PROGRAM INDEXING_2
VAR
	bStartInput : BOOL;
	bServoOn : BOOL;
	bProgram0_On : BOOL;
	bProgram1_On : BOOL :=TRUE;
	bProgram2_On : BOOL :=FALSE;
	bProgram3_On : BOOL:=FALSE;
	bProgram4_On : BOOL:=FALSE;	
	bHomePositionReturn : BOOL;
	bResetInput : BOOL;
	bEmergencyInput : BOOL := TRUE;
	
	IN_POSITION_INPUT: BOOL;
	IN_POSITIONING_COMPLETION: BOOL;
	IN_START_INPUT_WAIT: BOOL;
	IN_ALARM1: BOOL;
	IN_ALARM2: BOOL;
	IN_READY_STATE: BOOL;
	T1: TON;
	TMR1: TON;
	TMR2: TON;
	TMR3: TON;
	TMR4: TON;
	TMR5: TON;
	TMR6: TON;
	TMR7: TON;
	IN_SERVO_STATUS: BOOL;
	CNT1: CTU;
	ENABLE_TIMER: INT;
	ResetCount: BOOL;
	CNT_INDEX: CTU;
	
	RESET_CNT_INDEX: BOOL;
	TMR8: TON;
	M1:BOOL;
	M2:BOOL;
	M3:BOOL;
	M4:BOOL;
	TMR_OFF: TON;
	TMR_RELEASE: TON;
	IDX: INT;
END_VAR

VAR CONSTANT
	ISP: R_TRIG;
END_VAR

INDEXING_2_VAR.DataByteOutput2[0].0 := bProgram0_On;
INDEXING_2_VAR.DataByteOutput2[0].1 := bProgram1_On;
INDEXING_2_VAR.DataByteOutput2[0].2 := bProgram2_On;
INDEXING_2_VAR.DataByteOutput2[0].3 := bProgram3_On;
INDEXING_2_VAR.DataByteOutput2[0].4 := bProgram4_On;
INDEXING_2_VAR.DataByteOutput2[0].6 := bResetInput;
INDEXING_2_VAR.DataByteOutput2[0].7 := bHomePositionReturn;
INDEXING_2_VAR.DataByteOutput2[1].0 := bStartInput;
INDEXING_2_VAR.DataByteOutput2[1].1 := bServoOn;
INDEXING_2_VAR.DataByteOutput2[1].4 := bEmergencyInput;

IN_POSITION_INPUT := INDEXING_2_VAR.DataByteInput2 [1].0;
IN_POSITIONING_COMPLETION := INDEXING_2_VAR.DataByteInput2 [1].1;
IN_START_INPUT_WAIT := INDEXING_2_VAR.DataByteInput2 [1].2;
IN_ALARM1 := INDEXING_2_VAR.DataByteInput2 [1].3;
IN_ALARM2 := INDEXING_2_VAR.DataByteInput2 [1].4;
IN_READY_STATE :=INDEXING_2_VAR.DataByteInput2 [1].7;
IN_SERVO_STATUS :=INDEXING_2_VAR.DataByteInput2 [1].6; 

M1:=INDEXING_2_VAR.DataByteInput2 [0].0;
M2:=INDEXING_2_VAR.DataByteInput2 [0].1;
M3:=INDEXING_2_VAR.DataByteInput2 [0].2;
M4:=INDEXING_2_VAR.DataByteInput2 [0].3;
bProgram1_On:=FALSE;
bProgram2_On:=FALSE;
bProgram3_On:=FALSE;
bProgram4_On:=FALSE;

//CEK SERVO STATUS
IF NOT IN_SERVO_STATUS THEN
	bResetInput := TRUE;
	TMR4(IN:=bResetInput,PT:=T#0.5S);
	IF TMR4.Q THEN
		bResetInput := FALSE;
	END_IF
	bServoOn:=TRUE;
	//POWER_CONTROL.O_PWR_CTRL_INDEXING_2:=TRUE;
	TMR8(IN:=POWER_CONTROL.O_PWR_CTRL_INDEXING_2,PT:=T#0.5S);	
	IF TMR8.Q THEN
		POWER_CONTROL.O_PWR_CTRL_INDEXING_2:=FALSE;
		TMR8(IN:=FALSE);
	END_IF
END_IF

//ALARM RESET
IF NOT IN_ALARM1 OR NOT IN_ALARM2 THEN
	bResetInput := TRUE;
	TMR4(IN:=bResetInput,PT:=T#0.5S);
		INPUT_VAR.ALARM1:=NOT IN_ALARM1 OR NOT IN_ALARM2;
	IF TMR4.Q THEN
		bResetInput := FALSE;
	END_IF
ELSE
	TMR4(IN:=FALSE);
END_IF

//HOMING
IF NOT INDEXING_2_VAR.I_INDEXING_2_HOME THEN
 	INDEXING_2_VAR.O_INDEXING_HOME:=TRUE;
END_IF
 
IF INDEXING_2_VAR.O_INDEXING_HOME THEN
	bHomePositionReturn:=TRUE;
	ResetCount:=TRUE;
	INDEXING_2_VAR.I_INDEXING_2_ROTATION_DONE:=FALSE;
	RESET_CNT_INDEX:=TRUE;
ELSE
	RESET_CNT_INDEX:=FALSE;
	bHomePositionReturn:=FALSE;
END_IF

ISP(CLK:=IN_POSITIONING_COMPLETION);	
IF 	ISP.Q THEN
	INDEXING_2_VAR.I_INDEXING_2_ROTATION_DONE:=TRUE;
END_IF

IF INDEXING_2_VAR.I_INDEXING_2_ROTATION_DONE OR INDEXING_2_VAR.O_ROTATION_DONE THEN
	INDEXING_2_VAR.I_INDEXING_2_HOME:=TRUE;
	INDEXING_2_VAR.O_INDEXING_HOME:=FALSE;
END_IF
//POWER RESET
IF bHomePositionReturn OR NOT INDEXING_2_VAR.I_INDEXING_2_ROTATION_DONE THEN
	TMR_OFF(IN:=TRUE,PT:=T#60S);
	IF TMR_OFF.Q THEN
		POWER_CONTROL.O_PWR_CTRL_INDEXING_2:=TRUE;
		TMR_RELEASE(IN:=TRUE,PT:=T#0.5S);
		BPROGRAM0_ON:=FALSE;
	END_IF
ELSE
	TMR_OFF(IN:=FALSE);
	TMR_RELEASE(IN:=FALSE);
END_IF

IF TMR_RELEASE.Q THEN
	POWER_CONTROL.O_PWR_CTRL_INDEXING_1:=FALSE;
	TMR_OFF(IN:=FALSE);
END_IF



//START ROTATION 
	IF 	INDEXING_2_VAR.O_ROTATION_START AND IN_START_INPUT_WAIT AND NOT INDEXING_2_VAR.O_INDEXING_HOME THEN
		IDX:=1;
		INDEXING_2_VAR.I_INDEXING_2_ROTATION_DONE:=FALSE;
	END_IF
CASE IDX OF
1:
	bprogram0_on:=TRUE;
	IF BPROGRAM0_ON THEN
		IDX:=2;
		INDEXING_2_VAR.O_ROTATION_START:=FALSE;
	END_IF

2:
//select Program No.
	IF bprogram0_on THEN
		INDEXING_2_VAR.O_ROTATION_START:=FALSE;
		INDEXING_2_VAR.I_INDEXING_2_ROTATION_DONE:=FALSE;
		TMR1(IN:=bprogram0_on,PT:=T#15MS);
		bStartInput:=tmr1.Q ;
		IF tmr1.Q THEN
			TMR2(in:=TRUE,pt:=T#25MS);
		END_IF
	
		IF tmr2.Q THEN
			tmr1(in:=FALSE);
			bStartInput:=FALSE;
		END_IF
		tmr3(in:=tmr2.Q,pt:=T#5MS);
		IF tmr3.Q THEN
			bprogram0_on:= FALSE;
			tmr2(in:=FALSE);
			tmr3(in:=FALSE);
			
		END_IF
	END_IF
	IF 	ISP.Q THEN
		INDEXING_2_VAR.O_ROTATION_DONE:=TRUE;
		INDEXING_2_VAR.O_ROTATION_START:=FALSE;
		INDEXING_2_VAR.I_INDEXING_2_ROTATION_DONE:=TRUE;
		IDX:=3;
	END_IF
3:
		IF INDEXING_2_VAR.I_INDEXING_2_ROTATION_DONE OR INDEXING_2_VAR.O_ROTATION_DONE THEN
		IDX:=0;
	END_IF	
END_CASE


IF  INDEXING_2_VAR.I_INDEXING_2_HOME THEN
	CNT_INDEX(CU:=bprogram0_on,RESET:=CNT_INDEX.Q,PV:=4);
	ELSE
	CNT_INDEX(CU:=FALSE);
	INDEXING_2_VAR.CARRIER_INDEX :=100;
END_IF

CASE CNT_INDEX.CV OF
	0:
	INDEXING_2_VAR.CARRIER_INDEX :=0;
	RESET_CNT_INDEX:=FALSE;
	1:
	INDEXING_2_VAR.CARRIER_INDEX :=1;
	2:
	INDEXING_2_VAR.CARRIER_INDEX :=2;
	3:
	INDEXING_2_VAR.CARRIER_INDEX :=3;
ELSE
	INDEXING_2_VAR.CARRIER_INDEX :=0;
END_CASE

IF RESET_CNT_INDEX THEN
	CNT_INDEX(CU:=FALSE);
END_IF
//START ROTATING TRIGGER BY 3 ROBOTS
IF (TESTER_C8_VAR.READY_INDEXING AND LOADER_RS4_VAR.READY_INDEXING AND SORTER_RS4_VAR.READY_INDEXING)
	OR (LOADER_RS4_VAR.READY_INDEXING AND NOT TESTER_C8_VAR.O_C8_ENABLE)
	OR (TESTER_C8_VAR.READY_INDEXING AND LOADER_RS4_VAR.READY_INDEXING AND NOT SORTER_RS4_VAR.I_SORTER_RS4_ENABLE) THEN
	INDEXING_2_VAR.O_ROTATION_START:=TRUE;
ELSE
	INDEXING_2_VAR.O_ROTATION_START:=FALSE;
END_IF

END_PROGRAM

(* stored: Version 1.1.0.1, ProductVersion 3.1.4020.12
   POU INDEXING_2: Id {55c1d41c-bec4-4f85-b013-949698a43a00}, SpecialFunc None *)
